Staubli VAL3: selectType.pgx

program selectType()
  local string l_sMessage
  local num l_nIndex
  local string l_sEvent
  local num l_nDefault
  local num l_nKey
  local num i
  local string l_sPath
  local num l_nResult
begin
  // change the program type
  call use:clear(0,13)
  call language:message(l_sMessage,191)
  call use:typeCenter(13,l_sMessage,40,true)
  call use:setSizeList(10,2,15,6)
  // insert all the prog type list
  call use:listcreate("")
  call language:message(l_sMessage,25)
  call use:listadd(l_sMessage)
  l_sMessage="SUB-PROG"
  call use:listadd(l_sMessage)
  call language:message(l_sMessage,26)
  call use:listadd(l_sMessage)
  call use:selectNewField(nProgID,0,0)
  // select the Item
  do
    l_nKey=get()
    call use:listevent(l_nKey,l_nIndex,l_sEvent)
  until l_nKey==270 or l_nKey==255
  if l_nKey==270
    nProgID=l_nIndex
    if nProgID!=2
      sProgType=saveData:sProgType[nProgID]
    else
      // maintenance program
      sProgType=saveData:sProgType[0]
    endIf
    // load the progType
    call load()
    // rebuild the list
    call buildList()
    // refresh
    use:bUseRefresh=true
  endIf
end
